FUNCTION_BLOCK AxisJogTestSuite
VAR
	StubAxis : AXIS_REF;
	iStubTask : I_Task;
	TestAxisJog : JogTask := (AxisRef := stubaxis);
	ObjTestSuite : TestSuite<TestSuiteParameter.MaxTestCount>('C:\ProgramData\Beckhoff\TwinCAT\3.1\Boot\Object_Tests.xml') := (TestSuiteName := 'Object Test Suite');
END_VAR

DoesTaskAcceptAcceleration_Test();
DoesTaskAcceptDeceleration_Test();
DoesTaskAcceptJerk_Test();
DoesTaskAcceptsInch_Test();
DoesTaskRejectNegativeAccell_Test();
DoesTaskRejectNegativeDecel_Test();
DoesTaskRejectNegativeJerk_Test();
DoesTaskRejectZeroDistanceInch_Test();

METHOD DoesTaskAcceptAcceleration_Test
VAR_INST
	Expected : BOOL := TRUE;
	Actual	 : BOOL;
END_VAR
IF ObjTestSuite.Test(__POUNAME()).ExecuteTest() THEN
	TestAxisJog.Acceleration := 1.0;
	Actual := TestAxisJog.Acceleration = 1.0;
	ObjTestSuite.Test(__POUNAME()).AssertEqual(Expected, Actual);
	TestAxisJog.Acceleration := 0.0;
	TestAxisJog.Abort();
END_IF
END_METHOD

METHOD DoesTaskAcceptDeceleration_Test
VAR_INST
	Expected : BOOL := TRUE;
	Actual	 : BOOL;
END_VAR
IF ObjTestSuite.Test(__POUNAME()).ExecuteTest() THEN
	TestAxisJog.Deceleration := 1.0;
	Actual := TestAxisJog.Deceleration = 1.0;
	ObjTestSuite.Test(__POUNAME()).AssertEqual(Expected, Actual);
	TestAxisJog.Deceleration := 0.0;
	TestAxisJog.Abort();
END_IF
END_METHOD

METHOD DoesTaskAcceptJerk_Test
VAR_INST
	Expected : BOOL := TRUE;
	Actual	 : BOOL;
END_VAR
IF ObjTestSuite.Test(__POUNAME()).ExecuteTest() THEN
	TestAxisJog.Jerk := 1.0;
	Actual := TestAxisJog.Jerk = 1.0;
	ObjTestSuite.Test(__POUNAME()).AssertEqual(Expected, Actual);
	TestAxisJog.Jerk := 0.0;
	TestAxisJog.Abort();
END_IF
END_METHOD

METHOD DoesTaskAcceptsInch_Test
VAR_INST
	Expected : BOOL := TRUE;
	Actual	 : BOOL;
END_VAR
IF ObjTestSuite.Test(__POUNAME()).ExecuteTest() THEN
	Actual := SUCCEEDED(TestAxisJog.Inch(10.0,TRUE));
	ObjTestSuite.Test(__POUNAME()).AssertEqual(Expected, Actual);
	TestAxisJog.Abort();
END_IF
END_METHOD

METHOD DoesTaskRejectNegativeAccell_Test
VAR_INST
	Expected : BOOL := TRUE;
	Actual	 : BOOL;
END_VAR
IF ObjTestSuite.Test(__POUNAME()).ExecuteTest() THEN
	TestAxisJog.Acceleration := -1.0;
	Actual := TestAxisJog.Acceleration = 0.0;
	ObjTestSuite.Test(__POUNAME()).AssertEqual(Expected, Actual);
	TestAxisJog.Abort();
END_IF
END_METHOD

METHOD DoesTaskRejectNegativeDecel_Test
VAR_INST
	Expected : BOOL := TRUE;
	Actual	 : BOOL;
END_VAR
IF ObjTestSuite.Test(__POUNAME()).ExecuteTest() THEN
	TestAxisJog.Deceleration := -1.0;
	Actual := TestAxisJog.Deceleration = 0.0;
	ObjTestSuite.Test(__POUNAME()).AssertEqual(Expected, Actual);
	TestAxisJog.Abort();
END_IF
END_METHOD

METHOD DoesTaskRejectNegativeJerk_Test
VAR_INST
	Expected : BOOL := TRUE;
	Actual	 : BOOL;
END_VAR
IF ObjTestSuite.Test(__POUNAME()).ExecuteTest() THEN
	TestAxisJog.Jerk := -1.0;
	Actual := TestAxisJog.jerk = 0.0;
	ObjTestSuite.Test(__POUNAME()).AssertEqual(Expected, Actual);
	TestAxisJog.Abort();
END_IF
END_METHOD

METHOD DoesTaskRejectZeroDistanceInch_Test
VAR_INST
	Expected : BOOL := TRUE;
	Actual	 : BOOL;
END_VAR
IF ObjTestSuite.Test(__POUNAME()).ExecuteTest() THEN
	Actual := FAILED(TestAxisJog.Inch(-10.0,TRUE));
	ObjTestSuite.Test(__POUNAME()).AssertEqual(Expected, Actual);
	TestAxisJog.Abort();
END_IF
END_METHOD

END_FUNCTION_BLOCK

(* stored: Version 1.1.0.1
   POU AxisJogTestSuite: Id {d58fdfa9-a16a-4795-9564-e1d5a0ea8323}, SpecialFunc None
   Method DoesTaskAcceptAcceleration_Test: Id {97fe4398-d4c0-4835-9bd5-3582499aa884}
   Method DoesTaskAcceptDeceleration_Test: Id {716e911b-9a6c-4b43-bbeb-ede88198f42d}
   Method DoesTaskAcceptJerk_Test: Id {79558f02-1c76-467a-a708-5ab8b49e1f27}
   Method DoesTaskAcceptsInch_Test: Id {b603a83d-e08e-45f3-86b4-49fa0ebe0e9d}
   Method DoesTaskRejectNegativeAccell_Test: Id {4fe7aa44-c6df-45f2-9ce2-f90ef01c02cd}
   Method DoesTaskRejectNegativeDecel_Test: Id {2295c37c-d34d-4773-bd8b-50c76e582d1a}
   Method DoesTaskRejectNegativeJerk_Test: Id {7b320684-ada6-4bef-9fe2-3201a14cc365}
   Method DoesTaskRejectZeroDistanceInch_Test: Id {936752e7-1a5f-43db-9d36-dba5840b59e5} *)
